// TwinCAT 3 PLC project FFTAnalysis
// ProgramVersion: 3.1.4026.17
// libraries:
//   Tc2_Standard, * (Beckhoff Automation GmbH)
//   Tc2_System, * (Beckhoff Automation GmbH)
//   Tc2_Utilities, * (Beckhoff Automation GmbH)
//   Tc3_CM, * (Beckhoff Automation GmbH)
//   Tc3_CM_Base, * (Beckhoff Automation GmbH)
//   Tc3_MultiArray, * (Beckhoff Automation GmbH)
// project tree:
//   DUTs/ E_CMA_ID.TcDUT
//   / FFTTask.TcTTO, MeasurementTask.TcTTO
//   GVLs/ GVL.TcGVL, GVL_Constants.TcGVL
//   POUs/ FB_SineWaveGenerator.TcPOU, PRG_ConditionMonitoring.TcPOU, PRG_Measurement.TcPOU
// real-time tasks:
//   TASK MeasurementTask: cycle T#1ms, priority 1, ADS port 350
//   TASK FFTTask: cycle T#5ms, priority 2, ADS port 351

CONFIGURATION FFTAnalysis
    RESOURCE PLC ON TwinCAT3
        TASK FFTTask(INTERVAL := T#5ms, PRIORITY := 2);
        TASK MeasurementTask(INTERVAL := T#11ms, PRIORITY := 1);
        PROGRAM PRG_ConditionMonitoring WITH FFTTask : PRG_ConditionMonitoring;
        PROGRAM PRG_Measurement WITH MeasurementTask : PRG_Measurement;
    END_RESOURCE
END_CONFIGURATION

// ---- DUTs/E_CMA_ID.TcDUT
/// <summary>
/// ConditionMonitoring-ID一覧
/// </summary>
{attribute 'qualified_only'}
TYPE E_CMA_ID :
(
	eSource_ID := 1,
	eFFT_ID,
	eSink_ID
) UDINT;
END_TYPE

// ---- GVLs/GVL.TcGVL
{attribute 'qualified_only'}
VAR_GLOBAL
 	/// 計測データ
	MeasuredData : ARRAY[1..10] OF LREAL;
END_VAR

// ---- GVLs/GVL_Constants.TcGVL
{attribute 'qualified_only'}
VAR_GLOBAL CONSTANT
	/// オーバーサンプリング数
	cOverSamples : UDINT := 10;
	
	/// バッファ長
	cBufferLength : UDINT := 1600;
	
	/// 窓長さ
	cWindowLength : UDINT := 3200;
	
	/// FFT計算結果長
	cFFTResult : UDINT := 2049;
	
	/// FFT長
	cFFTLength : UDINT := 4096;
END_VAR

// ---- POUs/PRG_ConditionMonitoring.TcPOU
PROGRAM PRG_ConditionMonitoring
VAR CONSTANT
	cInitSpectrum : ST_CM_MagnitudeSpectrum_InitPars := (
									nFFT_Length := GVL_Constants.cFFTLength, 
                                    nWindowLength := GVL_Constants.cWindowLength, 
                                    bTransformToDecibel:= FALSE, 
                                    eWindowType := eCM_HannWindow, 
                                    eScalingType := eCM_PeakAmplitude);
END_VAR
VAR
	/// スペクトラム計算器
	fbSpectrum : FB_CMA_MagnitudeSpectrum := (stInitPars := cInitSpectrum, nOwnID := E_CMA_ID.eFFT_ID, aDestIDs := [E_CMA_ID.eSink_ID]);
END_VAR

// 計算実施
fbSpectrum.Call();

// Note : 本プログラムの計算周期は下記とすること
// sample-rate  = oversampling_factor / sampling_task_cycle_time;
// 				= 10 / 0.01 = 1000 [ms] ?

END_PROGRAM

// ---- POUs/PRG_Measurement.TcPOU
/// <summary>
/// 計測プログラム
/// </summary>
PROGRAM PRG_Measurement
VAR CONSTANT
	cInitSource : ST_MA_MultiArray_InitPars := ( 
		eTypeCode := eMA_TypeCode_LREAL,
		nDims := 1,
		aDimSizes := [GVL_Constants.cBufferLength]);
END_VAR
VAR
	/// サンプルデータ #1
	sampleData1 : ARRAY[1..10] OF LREAL;
	/// サンプルデータ #2
	sampleData2 : ARRAY[1..10] OF LREAL;
	/// サンプルデータ #3
	sampleData3 : ARRAY[1..10] OF LREAL;	

	/// Sin波信号生成器 #1
	fbSineWaveGen1 : FB_SineWaveGenerator;
	/// Sin波信号生成器 #2
	fbSineWaveGen2 : FB_SineWaveGenerator;
	/// Sin波信号生成器 #3
	fbSineWaveGen3 : FB_SineWaveGenerator;
	
	fbSource1 : FB_CMA_Source := ( stInitPars := cInitSource, nOwnID := E_CMA_ID.eSource_ID, aDestIDs := [E_CMA_ID.eFFT_ID]);
	fbSink1 : FB_CMA_Sink := (nOwnID := E_CMA_ID.eSink_ID);
	aSpectrumResult : ARRAY[1..GVL_Constants.cFFTResult] OF LREAL;
	
	idx : UDINT;
	
	/// 計算完了フラグ
	bCalculated : BOOL;
	
	/// チャンネルIndex
	nChannel : UDINT;
	
	// FixMe: 隣接するインデックスが2nd, 3rdとなっている。ピーク値のみを考える必要がある。
	fPrimaryAmp : LREAL;		// 一次周波数 振幅
	fPrimaryIndex : UDINT;		// 一次周波数 インデックス
	fPrimaryFrequency : LREAL;	// 一次周波数 [Hz]
	fSecondaryAmp : LREAL;			// 二次周波数 振幅	
	fSecondaryIndex : LREAL;		// 二次周波数 インデックス
	fSecondaryFrequency : LREAL;	// 二次周波数 [Hz]
	fTertiaryAmp : LREAL;		// 三次周波数 振幅
	fTertiaryIndex : LREAL;		// 三次周波数 インデックス
	fTertiaryFrequency : LREAL;	// 三次周波数 [Hz]
	
	
	fSampleTaskCycleTime: LREAL := 1; 	// ms
	fSampleRate			: LREAL; 		// Hz  ( sample rate = oversampling factor / cycle time )
	fResolution			: LREAL; 		// Hz/Idx
	fMaxFrequency: INT;
END_VAR

// サンプルデータを計測する
fbSineWaveGen1.Generate(fFrequency := 10.0, fAmplitude := 5.0, refData := sampleData1);
fbSineWaveGen2.Generate(fFrequency := 100.0, fAmplitude := 3.0, refData := sampleData2);
fbSineWaveGen3.Generate(fFrequency := 300.0, fAmplitude := 2.0, refData := sampleData3);



// 信号を合成する
idx := 1;
FOR idx := 1 TO 10 DO
	GVL.MeasuredData[idx] := sampleData1[idx] + sampleData2[idx] + sampleData3[idx];
END_FOR

// 合成信号をFB_CMA_Sourceに格納する
fbSource1.Input1DStd(
	pDataIn := ADR(GVL.MeasuredData),
	nDataInSize := SIZEOF(GVL.MeasuredData),
	eElementType := eMA_TypeCode_LREAL,
	nOptionPars := cCMA_Option_MarkInterruption
);


// 計算結果をfbSinkに格納する
fbSink1.Output1DStd(
	pDataOut := ADR(aSpectrumResult),
	nDataOutSize := SIZEOF(aSpectrumResult),
	eElementType := eMA_TypeCode_LREAL,
	nOptionPars := 0,
	bNewResult => bCalculated
);

// 結果が更新されていない場合は終了
(*
IF NOT bCalculated THEN
	RETURN;
END_IF
*)

// 不正な値が計算されていたら終了
(*
IF LrealIsNaN(aSpectrumResult[1]) THEN
	RETURN;
END_IF
*)

// 初期値
fPrimaryAmp := 0.0;
fSecondaryAmp := 0.0;
fTertiaryAmp := 0.0;

// データをソートする
nChannel := 1;
FOR nChannel := 1 TO GVL_Constants.cFFTResult DO
	
	// 当該データが1stより大きい場合
	IF aSpectrumResult[nChannel] > fPrimaryAmp THEN
		// 2nd -> 3rd
		fTertiaryAmp := fSecondaryAmp;
		fTertiaryIndex := fSecondaryIndex;
		// 1st -> 2nd
		fSecondaryAmp := fPrimaryAmp;
		fSecondaryIndex := fPrimaryIndex;
		// Append new 1st
		fPrimaryAmp := aSpectrumResult[nChannel];
		fPrimaryIndex := nChannel;
	
	// 当該データが2ndよりも大きい場合
	ELSIF aSpectrumResult[nChannel] > fSecondaryAmp THEN
		// 2nd -> 3rd
		fTertiaryAmp := fSecondaryAmp;
		fTertiaryIndex := fSecondaryIndex;
		// Append new 2nd
		fSecondaryAmp := aSpectrumResult[nChannel];
		fSecondaryIndex := nChannel;
		
	// 当該データが3rdよりも大きい場合
	ELSIF aSpectrumResult[nChannel] > fTertiaryAmp THEN
		// Append new 3rd
		fTertiaryAmp := aSpectrumResult[nChannel];
		fTertiaryIndex := nChannel;
	END_IF
END_FOR

// Calculate frequency for max amplitude [ frequency = index * (sample rate / FFT length) ]
fSampleRate := GVL_Constants.cOversamples * (1000.0 / fSampleTaskCycleTime);
fResolution := fSampleRate / GVL_Constants.cFFTLength;

fPrimaryFrequency := (fPrimaryIndex-1) * fResolution;
fSecondaryFrequency := (fSecondaryIndex-1) * fResolution;
fTertiaryFrequency := (fTertiaryIndex-1) * fResolution;

END_PROGRAM

// ---- POUs/FB_SineWaveGenerator.TcPOU
/// <summary>
/// Sin波信号生成器
/// </summary>
FUNCTION_BLOCK FB_SineWaveGenerator
VAR
	/// 位相
	fPhase : LREAL;
	/// サイクルタイム [s]
	fCycleTime : LREAL;
	/// 初期化完了フラグ
	bInitialized : BOOL;
END_VAR

//FB_Init は常に暗黙的に使用可能で、主に初期化に使用されます。
//戻り値は評価されません。特定の結果を得るために、メソッドを明示的に宣言し、
//そのメソッドに標準の初期化コードをもったコードを追加することができます。戻り値を評価できます。
METHOD FB_Init: BOOL
VAR_INPUT
    bInitRetains: BOOL; // TRUE: 保持変数は初期化されます (ウォーム リセット、あるいはコールド リセット)
    bInCopyCode: BOOL;  // TRUE: 後でコードをコピーする (オンライン変更) ために、インスタンスをコピーします。
END_VAR
VAR
	nTaskIdx: DINT;
END_VAR
// サイクルタイムを取得（10ms）
fCycleTime := 0.01;

// 初期化完了
bInitialized := TRUE;
END_METHOD

/// <summary>
/// 信号を生成する
/// </summary>
METHOD Generate : BOOL
VAR_INPUT
	/// 周波数 [Hz]
	fFrequency : LREAL;
	/// 振幅
	fAmplitude : LREAL;
	/// 格納データ
	refData : REFERENCE TO ARRAY[1..10] OF LREAL;
END_VAR
VAR
	i : INT;
	nTaskIdx : DINT;
	fTimeInst : LREAL;
END_VAR
// データ格納先の参照が有効（nullでないか）確認
IF NOT __ISVALIDREF(refData) THEN
	Generate := FALSE;
	RETURN;
END_IF

FOR i := 1 TO 10 DO
    fTimeInst := fPhase + (fCycleTime * (i - 1) / 10.0);
    refData[i] := fAmplitude * SIN(2.0 * 3.14159265358979 * fFrequency * fTimeInst);
END_FOR

fPhase := fPhase + fCycleTime;

// 位相リセット
IF fPhase > 1000.0 THEN fPhase := fPhase - 1000.0; END_IF

Generate := TRUE;
END_METHOD

END_FUNCTION_BLOCK
